SUBAPPLICATION Uebung_031_AX (* LED Strip *)
  (* Standard: 61499-2; Description: Copyright (c) 2026 Meisterschulen am Ostbahnhof This program and the accompanying materials are made available under the terms of the Eclipse Public License 2.0 which is available at https://www.eclipse.org/legal/epl-2.0/ SPDX-License-Identifier: EPL-2.0 *)
  (* Version 1.0, 2026-09-09, Franz Höpfinger, Meisterschulen am Ostbahnhof, initial API and implementation and/or initial documentation *)
  PACKAGE Uebungen;
  IMPORT logiBUS::io::DI::logiBUS_DI::Input_I1;
  IMPORT logiBUS::io::DI::logiBUS_DI::Input_I2;
  IMPORT logiBUS::io::DI::logiBUS_DI_Events::BUTTON_SINGLE_CLICK;
  IMPORT logiBUS::io::DO_LED::LED_strip;
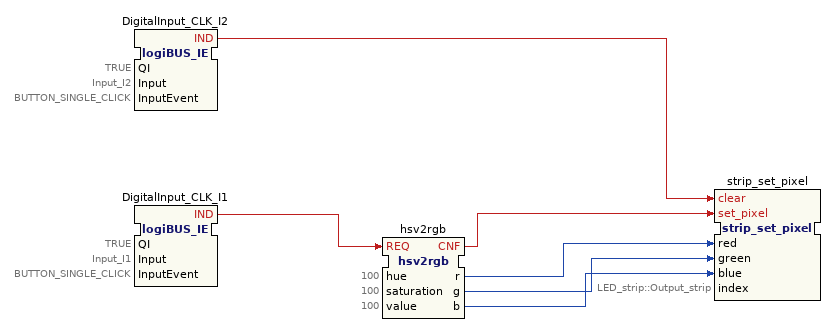
  FBS
    DigitalInput_CLK_I1 : logiBUS::io::DI::logiBUS_IE(QI := TRUE, Input := Input_I1, InputEvent := BUTTON_SINGLE_CLICK);
    DigitalInput_CLK_I2 : logiBUS::io::DI::logiBUS_IE(QI := TRUE, Input := Input_I2, InputEvent := BUTTON_SINGLE_CLICK);
    strip_set_pixel : logiBUS::esp32::rgb::strip_set_pixel(index := LED_strip::Output_strip);
    hsv2rgb : logiBUS::esp32::rgb::hsv2rgb(hue := 100, saturation := 100, value := 100);
  END_FBS
  EVENT_CONNECTIONS
    DigitalInput_CLK_I2.IND TO strip_set_pixel.clear;
    hsv2rgb.CNF TO strip_set_pixel.set_pixel;
    DigitalInput_CLK_I1.IND TO hsv2rgb.REQ;
  END_CONNECTIONS
  DATA_CONNECTIONS
    hsv2rgb.r TO strip_set_pixel.red;
    hsv2rgb.g TO strip_set_pixel.green;
    hsv2rgb.b TO strip_set_pixel.blue;
  END_CONNECTIONS
END_SUBAPPLICATION
